// TIA Portal V19 export
FUNCTION "RollformingMng_CALL" : Void   // FC164, LAD
TITLE = POST-PUNCHING MANAGER
// stored: SetENOAutomatically false
   VAR CONSTANT
      MIN_ROLLWAY_SPEED_RATIO : LReal := 150.0;
   END_VAR
BEGIN

REGION Network 1: Data In - Buttons
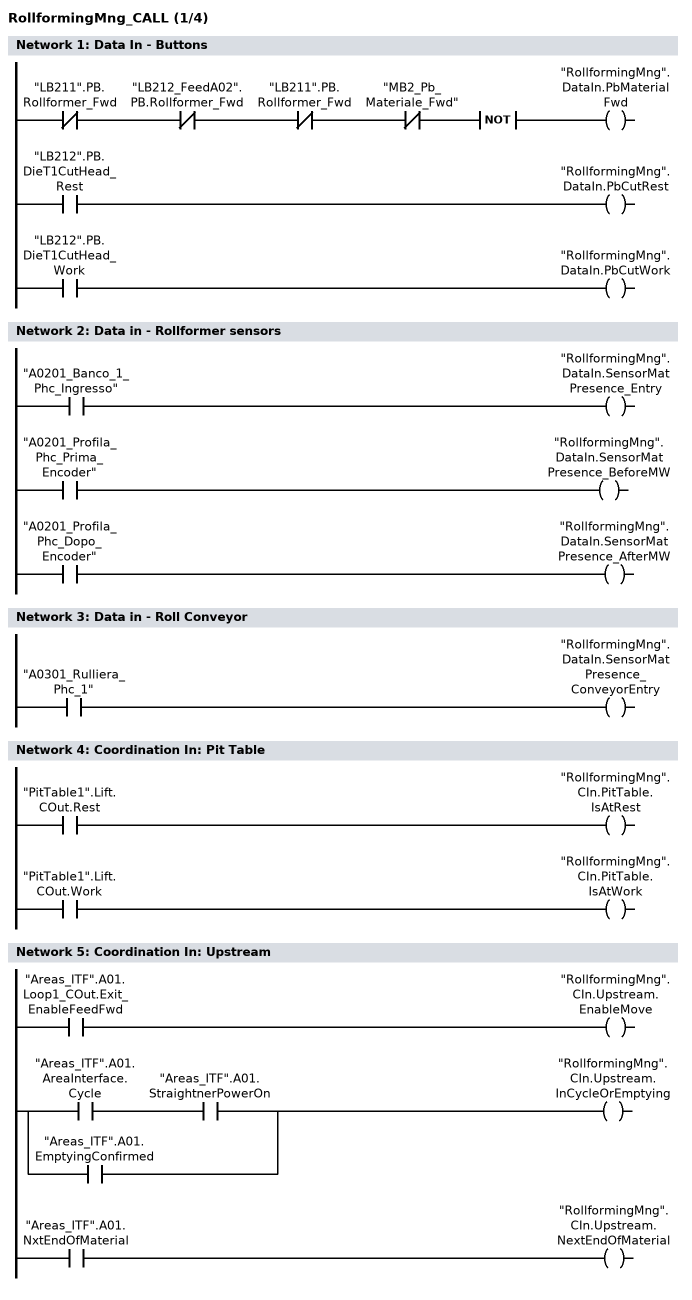
   RUNG wire#powerrail
      I_Contact( "LB211".PB.Rollformer_Fwd )
      I_Contact( "LB212_FeedA02".PB.Rollformer_Fwd )
      I_Contact( "LB211".PB.Rollformer_Fwd )
      I_Contact( "MB2_Pb_Materiale_Fwd" )
      Not()
      Coil( "RollformingMng".DataIn.PbMaterialFwd )
   END_RUNG
   RUNG wire#powerrail
      Contact( "LB212".PB.DieT1CutHead_Rest )
      Coil( "RollformingMng".DataIn.PbCutRest )
   END_RUNG
   RUNG wire#powerrail
      Contact( "LB212".PB.DieT1CutHead_Work )
      Coil( "RollformingMng".DataIn.PbCutWork )
   END_RUNG
   // the same network as SCL:
   "RollformingMng".DataIn.PbMaterialFwd := NOT (NOT "LB211".PB.Rollformer_Fwd AND NOT "LB212_FeedA02".PB.Rollformer_Fwd AND NOT "LB211".PB.Rollformer_Fwd AND NOT "MB2_Pb_Materiale_Fwd");
   "RollformingMng".DataIn.PbCutRest := "LB212".PB.DieT1CutHead_Rest;
   "RollformingMng".DataIn.PbCutWork := "LB212".PB.DieT1CutHead_Work;
END_REGION

REGION Network 2: Data in - Rollformer sensors
   RUNG wire#powerrail
      Contact( "A0201_Banco_1_Phc_Ingresso" )
      Coil( "RollformingMng".DataIn.SensorMatPresence_Entry )
   END_RUNG
   RUNG wire#powerrail
      Contact( "A0201_Profila_Phc_Prima_Encoder" )
      Coil( "RollformingMng".DataIn.SensorMatPresence_BeforeMW )
   END_RUNG
   RUNG wire#powerrail
      Contact( "A0201_Profila_Phc_Dopo_Encoder" )
      Coil( "RollformingMng".DataIn.SensorMatPresence_AfterMW )
   END_RUNG
   // the same network as SCL:
   "RollformingMng".DataIn.SensorMatPresence_Entry := "A0201_Banco_1_Phc_Ingresso";
   "RollformingMng".DataIn.SensorMatPresence_BeforeMW := "A0201_Profila_Phc_Prima_Encoder";
   "RollformingMng".DataIn.SensorMatPresence_AfterMW := "A0201_Profila_Phc_Dopo_Encoder";
END_REGION

REGION Network 3: Data in - Roll Conveyor
   RUNG wire#powerrail
      Contact( "A0301_Rulliera_Phc_1" )
      Coil( "RollformingMng".DataIn.SensorMatPresence_ConveyorEntry )
   END_RUNG
   // the same network as SCL:
   "RollformingMng".DataIn.SensorMatPresence_ConveyorEntry := "A0301_Rulliera_Phc_1";
END_REGION

REGION Network 4: Coordination In: Pit Table
   RUNG wire#powerrail
      Contact( "PitTable1".Lift.COut.Rest )
      Coil( "RollformingMng".CIn.PitTable.IsAtRest )
   END_RUNG
   RUNG wire#powerrail
      Contact( "PitTable1".Lift.COut.Work )
      Coil( "RollformingMng".CIn.PitTable.IsAtWork )
   END_RUNG
   // the same network as SCL:
   "RollformingMng".CIn.PitTable.IsAtRest := "PitTable1".Lift.COut.Rest;
   "RollformingMng".CIn.PitTable.IsAtWork := "PitTable1".Lift.COut.Work;
END_REGION

REGION Network 5: Coordination In: Upstream
   RUNG wire#powerrail
      Contact( "Areas_ITF".A01.Loop1_COut.Exit_EnableFeedFwd )
      Coil( "RollformingMng".CIn.Upstream.EnableMove )
   END_RUNG
   RUNG wire#powerrail
      Contact( "Areas_ITF".A01.AreaInterface.Cycle )
      Contact( "Areas_ITF".A01.StraightnerPowerOn )
      wire#w1
      Coil( "RollformingMng".CIn.Upstream.InCycleOrEmptying )
   END_RUNG
   RUNG wire#powerrail
      Contact( "Areas_ITF".A01.EmptyingConfirmed )
   END_RUNG wire#w1
   RUNG wire#powerrail
      Contact( "Areas_ITF".A01.NxtEndOfMaterial )
      Coil( "RollformingMng".CIn.Upstream.NextEndOfMaterial )
   END_RUNG
   // the same network as SCL:
   "RollformingMng".CIn.Upstream.EnableMove := "Areas_ITF".A01.Loop1_COut.Exit_EnableFeedFwd;
   "RollformingMng".CIn.Upstream.InCycleOrEmptying := ("Areas_ITF".A01.AreaInterface.Cycle AND "Areas_ITF".A01.StraightnerPowerOn) OR "Areas_ITF".A01.EmptyingConfirmed;
   "RollformingMng".CIn.Upstream.NextEndOfMaterial := "Areas_ITF".A01.NxtEndOfMaterial;
END_REGION

REGION Network 6: Coordination In - Profile program
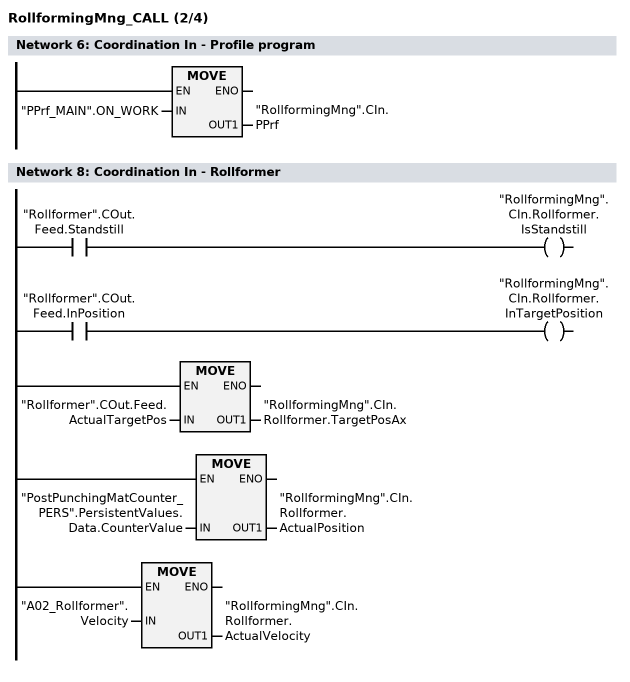
   RUNG wire#powerrail
      Move(in := "PPrf_MAIN".ON_WORK, out1 => "RollformingMng".CIn.PPrf)
   END_RUNG
   // the same network as SCL:
   "RollformingMng".CIn.PPrf := "PPrf_MAIN".ON_WORK;
END_REGION

REGION Network 7 (SCL): Coordination IN - Prod Manager
   "RollformingMng".CIn.ProdManager := "Areas_ITF".Prod.A02;
END_REGION

REGION Network 8: Coordination In - Rollformer
   RUNG wire#powerrail
      Contact( "Rollformer".COut.Feed.Standstill )
      Coil( "RollformingMng".CIn.Rollformer.IsStandstill )
   END_RUNG
   RUNG wire#powerrail
      Contact( "Rollformer".COut.Feed.InPosition )
      Coil( "RollformingMng".CIn.Rollformer.InTargetPosition )
   END_RUNG
   RUNG wire#powerrail
      { S7_GenerateENO := "TRUE" } Move(in := "Rollformer".COut.Feed.ActualTargetPos, out1 => "RollformingMng".CIn.Rollformer.TargetPosAx)
   END_RUNG
   RUNG wire#powerrail
      { S7_GenerateENO := "TRUE" } Move(in := "PostPunchingMatCounter_PERS".PersistentValues.Data.CounterValue, out1 => "RollformingMng".CIn.Rollformer.ActualPosition)
   END_RUNG
   RUNG wire#powerrail
      Move(in := "A02_Rollformer".Velocity, out1 => "RollformingMng".CIn.Rollformer.ActualVelocity)
   END_RUNG
   // the same network as SCL:
   "RollformingMng".CIn.Rollformer.IsStandstill := "Rollformer".COut.Feed.Standstill;
   "RollformingMng".CIn.Rollformer.InTargetPosition := "Rollformer".COut.Feed.InPosition;
   "RollformingMng".CIn.Rollformer.TargetPosAx := "Rollformer".COut.Feed.ActualTargetPos;
   "RollformingMng".CIn.Rollformer.ActualPosition := "PostPunchingMatCounter_PERS".PersistentValues.Data.CounterValue;
   "RollformingMng".CIn.Rollformer.ActualVelocity := "A02_Rollformer".Velocity;
END_REGION

REGION Network 9: Coordination In - Final Cut
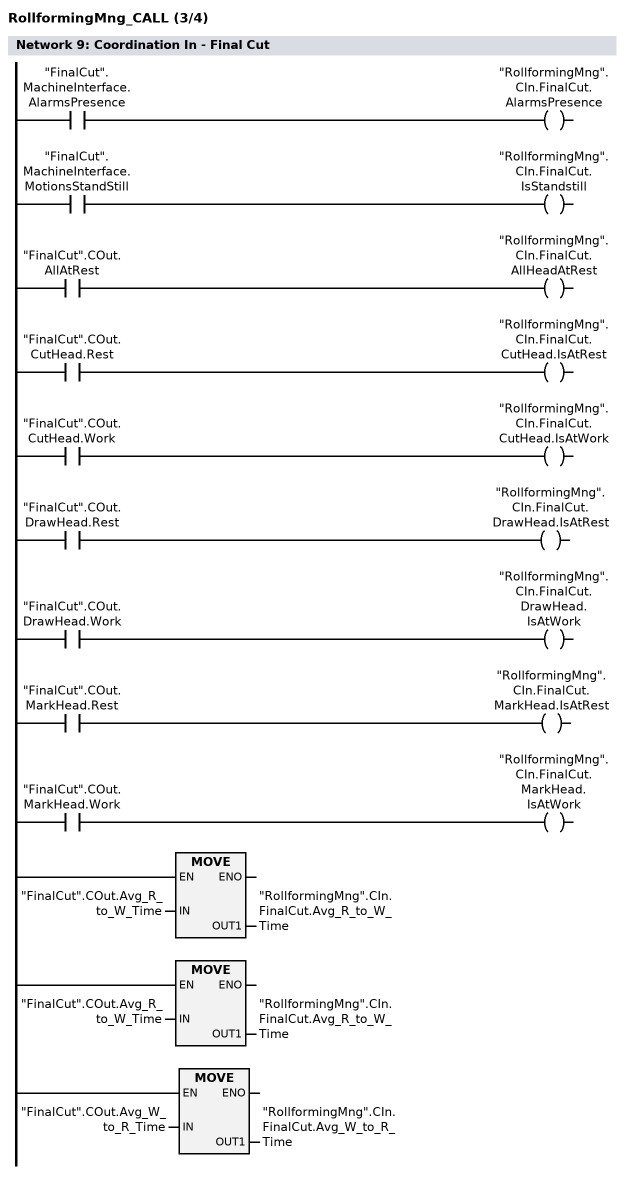
   RUNG wire#powerrail
      Contact( "FinalCut".MachineInterface.AlarmsPresence )
      Coil( "RollformingMng".CIn.FinalCut.AlarmsPresence )
   END_RUNG
   RUNG wire#powerrail
      Contact( "FinalCut".MachineInterface.MotionsStandStill )
      Coil( "RollformingMng".CIn.FinalCut.IsStandstill )
   END_RUNG
   RUNG wire#powerrail
      Contact( "FinalCut".COut.AllAtRest )
      Coil( "RollformingMng".CIn.FinalCut.AllHeadAtRest )
   END_RUNG
   RUNG wire#powerrail
      Contact( "FinalCut".COut.CutHead.Rest )
      Coil( "RollformingMng".CIn.FinalCut.CutHead.IsAtRest )
   END_RUNG
   RUNG wire#powerrail
      Contact( "FinalCut".COut.CutHead.Work )
      Coil( "RollformingMng".CIn.FinalCut.CutHead.IsAtWork )
   END_RUNG
   RUNG wire#powerrail
      Contact( "FinalCut".COut.DrawHead.Rest )
      Coil( "RollformingMng".CIn.FinalCut.DrawHead.IsAtRest )
   END_RUNG
   RUNG wire#powerrail
      Contact( "FinalCut".COut.DrawHead.Work )
      Coil( "RollformingMng".CIn.FinalCut.DrawHead.IsAtWork )
   END_RUNG
   RUNG wire#powerrail
      Contact( "FinalCut".COut.MarkHead.Rest )
      Coil( "RollformingMng".CIn.FinalCut.MarkHead.IsAtRest )
   END_RUNG
   RUNG wire#powerrail
      Contact( "FinalCut".COut.MarkHead.Work )
      Coil( "RollformingMng".CIn.FinalCut.MarkHead.IsAtWork )
   END_RUNG
   RUNG wire#powerrail
      Move(in := "FinalCut".COut.Avg_R_to_W_Time, out1 => "RollformingMng".CIn.FinalCut.Avg_R_to_W_Time)
   END_RUNG
   RUNG wire#powerrail
      Move(in := "FinalCut".COut.Avg_R_to_W_Time, out1 => "RollformingMng".CIn.FinalCut.Avg_R_to_W_Time)
   END_RUNG
   RUNG wire#powerrail
      Move(in := "FinalCut".COut.Avg_W_to_R_Time, out1 => "RollformingMng".CIn.FinalCut.Avg_W_to_R_Time)
   END_RUNG
   // the same network as SCL:
   "RollformingMng".CIn.FinalCut.AlarmsPresence := "FinalCut".MachineInterface.AlarmsPresence;
   "RollformingMng".CIn.FinalCut.IsStandstill := "FinalCut".MachineInterface.MotionsStandStill;
   "RollformingMng".CIn.FinalCut.AllHeadAtRest := "FinalCut".COut.AllAtRest;
   "RollformingMng".CIn.FinalCut.CutHead.IsAtRest := "FinalCut".COut.CutHead.Rest;
   "RollformingMng".CIn.FinalCut.CutHead.IsAtWork := "FinalCut".COut.CutHead.Work;
   "RollformingMng".CIn.FinalCut.DrawHead.IsAtRest := "FinalCut".COut.DrawHead.Rest;
   "RollformingMng".CIn.FinalCut.DrawHead.IsAtWork := "FinalCut".COut.DrawHead.Work;
   "RollformingMng".CIn.FinalCut.MarkHead.IsAtRest := "FinalCut".COut.MarkHead.Rest;
   "RollformingMng".CIn.FinalCut.MarkHead.IsAtWork := "FinalCut".COut.MarkHead.Work;
   "RollformingMng".CIn.FinalCut.Avg_R_to_W_Time := "FinalCut".COut.Avg_R_to_W_Time;
   "RollformingMng".CIn.FinalCut.Avg_R_to_W_Time := "FinalCut".COut.Avg_R_to_W_Time;
   "RollformingMng".CIn.FinalCut.Avg_W_to_R_Time := "FinalCut".COut.Avg_W_to_R_Time;
END_REGION

REGION Network 10: Coordination in - Material counter
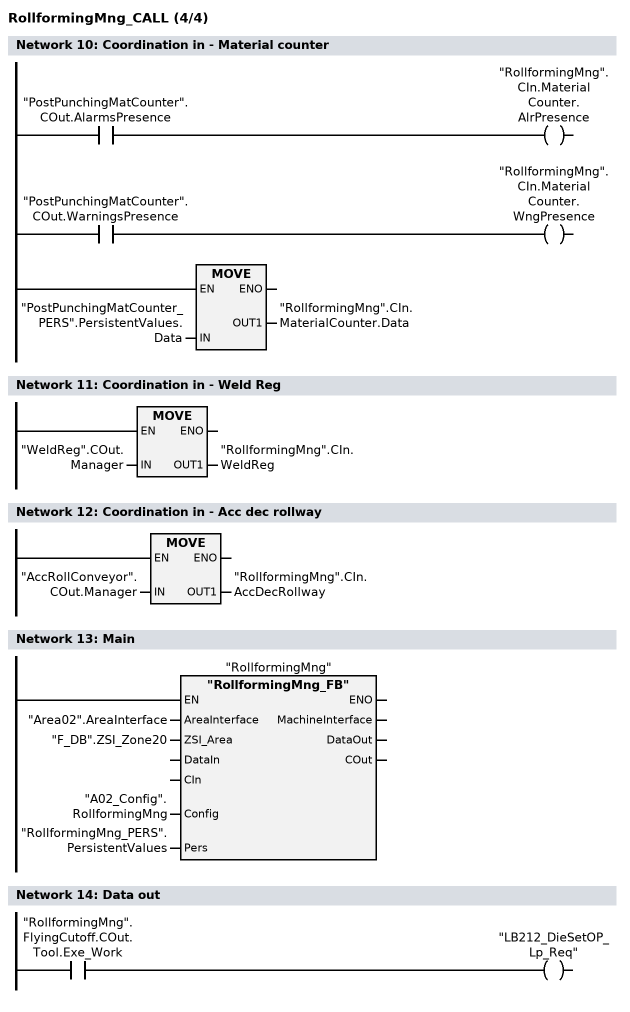
   RUNG wire#powerrail
      Contact( "PostPunchingMatCounter".COut.AlarmsPresence )
      Coil( "RollformingMng".CIn.MaterialCounter.AlrPresence )
   END_RUNG
   RUNG wire#powerrail
      Contact( "PostPunchingMatCounter".COut.WarningsPresence )
      Coil( "RollformingMng".CIn.MaterialCounter.WngPresence )
   END_RUNG
   RUNG wire#powerrail
      Move(in := "PostPunchingMatCounter_PERS".PersistentValues.Data, out1 => "RollformingMng".CIn.MaterialCounter.Data)
   END_RUNG
   // the same network as SCL:
   "RollformingMng".CIn.MaterialCounter.AlrPresence := "PostPunchingMatCounter".COut.AlarmsPresence;
   "RollformingMng".CIn.MaterialCounter.WngPresence := "PostPunchingMatCounter".COut.WarningsPresence;
   "RollformingMng".CIn.MaterialCounter.Data := "PostPunchingMatCounter_PERS".PersistentValues.Data;
END_REGION

REGION Network 11: Coordination in - Weld Reg
   RUNG wire#powerrail
      Move(in := "WeldReg".COut.Manager, out1 => "RollformingMng".CIn.WeldReg)
   END_RUNG
   // the same network as SCL:
   "RollformingMng".CIn.WeldReg := "WeldReg".COut.Manager;
END_REGION

REGION Network 12: Coordination in - Acc dec rollway
   RUNG wire#powerrail
      Move(in := "AccRollConveyor".COut.Manager, out1 => "RollformingMng".CIn.AccDecRollway)
   END_RUNG
   // the same network as SCL:
   "RollformingMng".CIn.AccDecRollway := "AccRollConveyor".COut.Manager;
END_REGION

REGION Network 13: Main
   RUNG wire#powerrail
      "RollformingMng"(AreaInterface := "Area02".AreaInterface, ZSI_Area := "F_DB".ZSI_Zone20, DataIn :=, CIn :=, Config := "A02_Config".RollformingMng, Pers := "RollformingMng_PERS".PersistentValues, MachineInterface =>, DataOut =>, COut =>)
   END_RUNG
   // the same network as SCL:
   "RollformingMng"(AreaInterface := "Area02".AreaInterface,   // "RollformingMng_FB"
                    ZSI_Area := "F_DB".ZSI_Zone20,
                    Config := "A02_Config".RollformingMng,
                    Pers := "RollformingMng_PERS".PersistentValues);
END_REGION

REGION Network 14: Data out
   RUNG wire#powerrail
      Contact( "RollformingMng".FlyingCutoff.COut.Tool.Exe_Work )
      Coil( "LB212_DieSetOP_Lp_Req" )
   END_RUNG
   // the same network as SCL:
   "LB212_DieSetOP_Lp_Req" := "RollformingMng".FlyingCutoff.COut.Tool.Exe_Work;
END_REGION
END_FUNCTION
